# B&R Automation Studio project MachineControl
Automation Studio 4.12.2.93

## Configuration Config1

### Hardware
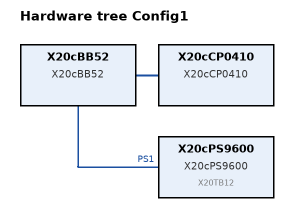
```
X20TB12 : X20TB12 v1.0.0.0
X20cBB52 : X20cBB52 v1.1.0.0
X20cCP0410 : X20cCP0410 v1.2.0.0  [SL -> X20cBB52.SL1]
  Connector IF2:
    ActivateDevice = 1
  ConfigurationID = MachineControl_Config1
  TimerDeviceType = SWIOTIMER
  Cyclic1Duration = 10000
  Cyclic1Tolerance = 10000
  Cyclic2Duration = 20000
  Cyclic2Tolerance = 20000
  Cyclic3Duration = 50000
  Cyclic3Tolerance = 50000
  Cyclic4Duration = 100000
  Cyclic4Tolerance = 100000
  Cyclic5Duration = 200000
  Cyclic5Tolerance = 200000
  Cyclic6Duration = 500000
  Cyclic6Tolerance = 500000
  Cyclic7Duration = 1000000
  Cyclic7Tolerance = 1000000
  Cyclic8Duration = 10000
  Cyclic8Tolerance = 30000000
  FileDevice1
  FileDeviceName1 = USER
  FileDevicePath1 = USER_PATH
X20cPS9600 : X20cPS9600 v1.2.1.0  [PS -> X20cBB52.PS1; SS1 -> X20TB12.SS]
```

## Logical view

### Global.typ
```iecst
(*//Pb Controll Start_							-1*)

TYPE
	tyPushButtonsControl : 	STRUCT
		Outputs : tyOutputs;
		Inputs : tyInputs;
		StaticVar : tyStatic;
	END_STRUCT;
	tyOutputs : 	STRUCT
		bGlobalReset : BOOL;
		bSystemInStopMode : BOOL;
		bSystemInRunMode : BOOL;
	END_STRUCT;
	tyInputs : 	STRUCT
		bResetPb : BOOL;
		bStopPb : BOOL;
		bRunPb : BOOL;
	END_STRUCT;
	tyStatic : 	STRUCT
		f_Trig_StopPb : f_trig;
		f_Trig_RunPb : f_trig;
	END_STRUCT;
END_TYPE

(*//Pb Controll End*)
```

### Global.var
```iecst
VAR
	DeviceModeControll : tyPushButtonsControl;
END_VAR
```

### Program Logical/Program

#### Cyclic.st
```iecst
PROGRAM _CYCLIC
//=============================================================================
// Dmitri Raihtsaum - Copyright 2023
// Created By: Dmitri Raihtsaum
//-----------------------------------------------------------------------------
// Tested with:   X20cCP0410
// Engineering:   Automation Studio 4.12
// Functionality: Machine controll pushbuttons logic for training
// Date: 17.03.2023
// Rev 0.1
//=============================================================================

	///Mapping
	DeviceModeControll.StaticVar.f_Trig_RunPb(CLK := DeviceModeControll.Inputs.bRunPb);
	DeviceModeControll.StaticVar.f_Trig_StopPb(CLK := DeviceModeControll.Inputs.bStopPb);

	//Protection
	IF DeviceModeControll.Outputs.bSystemInRunMode AND DeviceModeControll.Outputs.bSystemInStopMode THEN
		DeviceModeControll.Outputs.bSystemInStopMode :=TRUE;
		DeviceModeControll.Outputs.bSystemInRunMode :=FALSE;
		END_IF;
	IF NOT DeviceModeControll.Outputs.bSystemInRunMode AND NOT DeviceModeControll.Outputs.bSystemInStopMode THEN
		DeviceModeControll.Outputs.bSystemInStopMode :=TRUE;
		DeviceModeControll.Outputs.bSystemInRunMode :=FALSE;
	END_IF;
	//Code
	//Butons Control
	//Run button pressed
	IF DeviceModeControll.StaticVar.f_Trig_RunPb.Q THEN
		DeviceModeControll.Outputs.bSystemInStopMode :=FALSE;
		DeviceModeControll.Outputs.bSystemInRunMode :=TRUE;
	END_IF;
	//Stop button pressed
	IF DeviceModeControll.StaticVar.f_Trig_StopPb.Q THEN
		DeviceModeControll.Outputs.bSystemInStopMode :=TRUE;
		DeviceModeControll.Outputs.bSystemInRunMode :=FALSE;
	END_IF;
		//Global Reset can be pressed when system in stop mode
		IF DeviceModeControll.Outputs.bSystemInStopMode AND DeviceModeControll.Inputs.bResetPb THEN
		DeviceModeControll.Outputs.bGlobalReset :=TRUE;
	ELSE
		DeviceModeControll.Outputs.bGlobalReset :=FALSE;
	END_IF;

	//////////////////////////////////////// END ////////////////////////////////////////
END_PROGRAM
```

#### Init.st
```iecst
PROGRAM _INIT
	DeviceModeControll.Outputs.bSystemInRunMode :=FALSE;
	DeviceModeControll.Outputs.bSystemInStopMode :=TRUE;
	DeviceModeControll.StaticVar.f_Trig_RunPb.CLK := FALSE;
	DeviceModeControll.StaticVar.f_Trig_StopPb.CLK := FALSE;
END_PROGRAM
```
